PROGRAM Kollisionserkennung
VAR
	robotPoseArray AT%I*: ARRAY[1..8] OF RobotPose;
	robotPoseLokal : ARRAY[1..8] OF RobotPose;
	vxRobot AT%I*: LREAL;
	vyRobot AT%I*: LREAL;
	collisionDetected : BOOL := FALSE;
	robotCollision AT%Q* : ARRAY[0..4] OF BOOL;
		
	xRobot, yRobot: LREAL;
	i, j, k, l, m, n, o : INT := 1;
	quadrant : INT := 0;
	robotActive :ARRAY[1..4] OF INT;
	noCamera, cameraDown, permanentDown, stateCameraDown  : BOOL := FALSE;
	
	//Bounding Box
	x1Box,y1Box,x2Box,y2Box,x3Box,y3Box,x4Box,y4Box : LREAL; 
	alpha, beta, gamma, diagonal : LREAL := 0.0;
	breite, laenge : INT;
	
	//Timer
	timer :TON;
	timeValue : TIME := T#2S;
END_VAR

 timer(IN:= noCamera, PT := timeValue); //Roboter darf 2s blind fahren

//suche die Position des passenden Roboters
FOR i := 1 TO 4 BY 1 DO
	IF i = Var_HAWIno.Robot_Number THEN
		xRobot := robotPoseArray[i].x;
		yRobot := robotPoseArray[i].y;
	END_IF
END_FOR

//350mm Durchmesser des Roboters & 70mm Toleranzabstand
breite := 350 + 80; 
laenge := 350 + 80;
diagonal := SQRT(EXPT(breite,2) + EXPT(laenge,2));
IF vyRobot <> 0 AND vxRobot <> 0 THEN
	gamma  := ATAN2(vyRobot,vxRobot); //Drehung des Roboters
END_IF
beta := ATAN(laenge/breite); //Winkel des festen Dreiecks

//Kameradaten verfügbar 
IF xRobot <> 0 AND yRobot <> 0 THEN
	noCamera := FALSE;
	cameraDown := FALSE;
	
	//Zurücksetzen wenn Kameradaten wieder da
	IF stateCameraDown = TRUE THEN
		stateCameraDown := FALSE;
		FOR n:= 0 TO 4 BY 1 DO
			robotCollision[n] := FALSE;
		END_FOR
	END_IF
	
	//Zwischenspeicher der letzten Positionen wenn die Kameradaten ausfallen
	FOR m := 1 TO 8 BY 1 DO
		robotPoseLokal[m].x := robotPoseArray[m].x;
		robotPoseLokal[m].y := robotPoseArray[m].y;
		robotPoseLokal[m].theta := robotPoseArray[m].theta;
		robotPoseLokal[m].e := robotPoseArray[m].e;
	END_FOR
	
//Kameradaten ausfallen	
ELSE
	noCamera := TRUE;
	cameraDown := TRUE;
	//Kameradaten länger als 2s ausfallen, setzen die Array auf true
	IF timer.Q THEN
		permanentDown := TRUE;
	ELSE
		permanentDown := FALSE;
	END_IF
END_IF

//Kameradaten ausfallen, dann die lokale Position wird zugegriffen
IF cameraDown = TRUE AND permanentDown = FALSE THEN
	xRobot := robotPoseLokal[Var_HAWIno.Robot_Number].x;
	yRobot := robotPoseLokal[Var_HAWIno.Robot_Number].y;
	FOR l := 1 TO 8 BY 1 DO
		robotPoseArray[l].x := robotPoseLokal[l].x;
		robotPoseArray[l].y := robotPoseLokal[l].y;
		robotPoseArray[l].theta := robotPoseLokal[l].theta;
		robotPoseArray[l].e := robotPoseLokal[l].e;
	END_FOR
//Kameradaten 2s lang ausfallen, ist die gesamte Array True
ELSIF cameraDown = TRUE AND permanentDown = TRUE THEN
	xRobot := 0.0;
	yRobot := 0.0;
	FOR n:= 0 TO 4 BY 1 DO
		robotCollision[n] := TRUE;
	END_FOR
	stateCameraDown := TRUE;
END_IF

//Bounding Box dreht mit der Roboterblickrichtung
IF gamma >= 0 AND gamma < pi/2 THEN //Quadrant 1
	quadrant := 1;
	alpha := pi/2 - gamma; //Winkel des gedrehten Boxes
	x1Box := xRobot + COS(alpha) * breite;
	y1Box := yRobot - SIN(alpha) * breite;
	x2Box := xRobot + SIN(alpha + beta) * diagonal;
	y2Box := yRobot + COS(alpha + beta) * diagonal;
	x3Box := xRobot - COS(alpha + beta) * diagonal;
	y3Box := yRobot + SIN(alpha + beta) * diagonal;
	x4Box := xRobot - COS(alpha) * breite;
	y4Box := yRobot + SIN(alpha) * breite;	
ELSIF gamma >= pi/2 AND gamma <= pi THEN //Quadrant 2
	quadrant := 2;
	alpha := pi - gamma;
	x1Box := xRobot + SIN(alpha) * breite;
	y1Box := yRobot + COS(alpha) * breite;
	x2Box := xRobot - COS(alpha + beta) * diagonal;
	y2Box := yRobot + SIN(alpha + beta) * diagonal;
	x3Box := xRobot - SIN(alpha + beta) * diagonal;
	y3Box := yRobot - COS(alpha + beta) * diagonal;
	x4Box := xRobot - SIN(alpha) * breite;
	y4Box := yRobot - COS(alpha) * breite;
ELSIF gamma > -pi AND gamma < -pi/2 THEN //Quadrant 3
	quadrant := 3;
	alpha := pi + gamma;
	x1Box := xRobot - SIN(alpha) * breite;
	y1Box := yRobot + COS(alpha) * breite;
	x2Box := xRobot - SIN(alpha + beta) * diagonal;
	y2Box := yRobot + COS(alpha + beta) * diagonal;
	x3Box := xRobot - COS(alpha + beta) * diagonal;
	y3Box := yRobot - SIN(alpha + beta) * diagonal;
	x4Box := xRobot + SIN(alpha) * breite;
	y4Box := yRobot - COS(alpha) * breite;	
ELSIF gamma >= -pi/2 AND gamma < 0 THEN //Quadrant 4
	quadrant := 4;
	alpha := gamma + pi/2;
	x1Box := xRobot - COS(alpha) * breite;
	y1Box := yRobot - SIN(alpha) * breite;
	x2Box := xRobot - COS(alpha + beta) * diagonal;
	y2Box := yRobot - SIN(alpha + beta) * diagonal;
	x3Box := xRobot + SIN(alpha + beta) * diagonal;
	y3Box := yRobot - COS(alpha + beta) * diagonal;
	x4Box := xRobot + COS(alpha) * breite;
	y4Box := yRobot + SIN(alpha) * breite;
END_IF

//Finde alle aktiven Roboter im Feld
FOR j := 1 TO 4 BY 1 DO
	IF robotPoseArray[j].x <> 0 AND robotPoseArray[j].y <> 0 AND j <> Var_HAWIno.Robot_Number THEN
		robotActive[j] := j;
	END_IF
END_FOR

//Erkennt Roboter Kollision in Box?
FOR k := 1 TO 4 BY 1 DO
	IF robotActive [k] <> 0 AND robotActive [k] <> Var_HAWIno.Robot_Number THEN
		IF quadrant = 1 THEN
			IF robotPoseArray[robotActive[k]].x < x2Box AND robotPoseArray[robotActive[k]].x > x4Box AND robotPoseArray[robotActive[k]].y < y3Box AND robotPoseArray[robotActive[k]].y > y1Box THEN
				collisionDetected := TRUE;
			ELSE
				collisionDetected := FALSE;
			END_IF
		ELSIF quadrant = 2 THEN
			IF robotPoseArray[robotActive[k]].x < x1Box AND robotPoseArray[robotActive[k]].x > x3Box AND robotPoseArray[robotActive[k]].y < y2Box AND robotPoseArray[robotActive[k]].y > y4Box THEN
				collisionDetected := TRUE;
			ELSE
				collisionDetected := FALSE;
			END_IF
		ELSIF quadrant = 3 THEN
			IF robotPoseArray[robotActive[k]].x < x4Box AND robotPoseArray[robotActive[k]].x > x2Box AND robotPoseArray[robotActive[k]].y < y1Box AND robotPoseArray[robotActive[k]].y > y3Box THEN
				collisionDetected := TRUE;
			ELSE
				collisionDetected := FALSE;
			END_IF
		ELSIF quadrant = 4 THEN
			IF robotPoseArray[robotActive[k]].x < x3Box AND robotPoseArray[robotActive[k]].x > x1Box AND robotPoseArray[robotActive[k]].y < y4Box AND robotPoseArray[robotActive[k]].y > y2Box THEN
				collisionDetected := TRUE;
			ELSE
				collisionDetected := FALSE;
			END_IF
		END_IF
	END_IF
	
	IF collisionDetected = TRUE THEN
		robotCollision[robotActive[k]] := TRUE;
	ELSE 
		robotCollision[robotActive[k]] := FALSE;
	END_IF
END_FOR

END_PROGRAM

(* stored: Version 1.1.0.1, ProductVersion 3.1.4024.11
   POU Kollisionserkennung: Id {2163055e-1523-4ae1-8ad2-f781f29a50e9}, SpecialFunc None *)
